(* CODESYS project PlantaFinal.project

Project tree, tasks and I/O mapping:
  Device : CODESYS Control Win V3, 3S - Smart Software Solutions GmbH, order no. 305021, version 3.5.8.10
    application Application
      libraries: Standard, * (System)
      task MainTask (cyclic, interval t#20ms, priority 1) calls PLC_PRG
      program PLC_PRG [LD]
      Symbols
*)

// Device/Application/PLC_PRG
PROGRAM PLC_PRG
VAR
	//Entradas - Gerais
	_EmergencyStop: BOOL;
	_Reset: BOOL;
	_Start: BOOL;
	_Stop: BOOL;
	_Auto: BOOL;
	_Manual: BOOL;
	
	//Entradas - Stage 01
	_S01_VisionSensor1: WORD;
	_S01_VisionSensor2: WORD;	
	_S01_Sensor1: BOOL;
	_S01_Sensor2: BOOL;	
	_S01_Pusher1Back: BOOL;
	_S01_Pusher2Back: BOOL;	
	_S01_Pusher1Front: BOOL;
	_S01_Pusher2Front: BOOL;	
	_S01_AtPusher1Exit: BOOL;
	_S01_AtPusher2Exit: BOOL;
	_S01_LidAtExit: BOOL;
	_S01_BaseAtExit: BOOL;
	
	//Entradas - Stage 02
	_S02_LidAtEntry: BOOL;
	_S02_BaseAtEntry: BOOL;
	_S02_LidAtPlace: BOOL;
	_S02_LidClamped: BOOL;
	_S02_BaseClamped: BOOL;
	_S02_MovingZ: BOOL;
	_S02_BaseAtPlace: BOOL;
	_S02_MovingX: BOOL;
	_S02_PartLeaving: BOOL;
	
	//Entradas - Stage 03
	_S03_ItemAtEntry: BOOL;
	_S03_ItemADetected: BOOL;
	_S03_MovingX: BOOL;
	_S03_MovingZ: BOOL;
	
	//Entradas - Stage 04
	_S04_AtEntry: BOOL;
	_S04_AtLoad: BOOL;
	_S04_AtLeft: BOOL;
	_S04_AtRight: BOOL;
	_S04_AtMiddle: BOOL;
	_S04_MovingZ: BOOL;
	_S04_MovingX: BOOL;
	
	//Saidas - Gerais
	StopLight: BOOL;
	StartLight: BOOL;
	ResetLight: BOOL;
	ProductCounter: WORD;
	
	//Saidas - Stage 01
	S01_EntryConveyor1: BOOL;
	S01_EntryConveyor2: BOOL;
	S01_Conveyor1: BOOL;
	S01_Conveyor2: BOOL;
	S01_Pusher1: BOOL;
	S01_Pusher2: BOOL;
	S01_RollerStop1: BOOL;
	S01_RollerStop2: BOOL;
	
	//Saidas - Stage 02
	S02_LidsConveyor: BOOL;
	S02_BasesConveyor: BOOL;
	S02_ClampLid: BOOL;
	S02_MoveZ: BOOL;
	S02_MoveX: BOOL;
	S02_Grab: BOOL;
	S02_ClampBase: BOOL;
	S02_PosRaiseBase: BOOL;
	
	//Saidas - Stage 03
	S03_Grab: BOOL;
	S03_MoveZ: BOOL;
	S03_MoveX: BOOL;
	S03_EntryConveyor: BOOL;
	S03_Emitter: BOOL;
	S03_RollerConveyor: BOOL;

	//Saidas - Stage 03
	S04_EntryConveyor: BOOL;	
	S04_LoadConveyor: BOOL;
	S04_ForksLeft: BOOL;
	S04_ForksRight: BOOL;
	S04_Lift: BOOL;	
	S04_TargetPosition: INT;	
	
	//Sinais - Gerais
	Enable: BOOL;
	Stopping: BOOL;
	OnDelay: TON;
	OffDelay: TOF;
	AutoMode: BOOL;
	ManualMode: BOOL;	
	Caso: INT;	
	BaseAzul: WORD :=3;
	BaseVerde: WORD :=6;
	TampaAzul: WORD :=2;
	TampaVerde: WORD :=5;
	
	//Sinais - Stage 01
	S01_MX10: BOOL;
	S01_MX11: BOOL;
	S01_MX12: BOOL;
	S01_MX13: BOOL;
	S01_MX14: BOOL;
	S01_MX15: BOOL;
	S01_MX16: BOOL;
	S01_MX17: BOOL;
	F_TRIG_0: F_TRIG;
	F_TRIG_1: F_TRIG;
	F_TRIG_2: F_TRIG;
	F_TRIG_3: F_TRIG;
	F_TRIG_4: F_TRIG;	
	F_TRIG_5: F_TRIG;
	F_TRIG_6: F_TRIG;
	F_TRIG_7: F_TRIG;
	F_TRIG_8: F_TRIG;
	PartsAtExit: BOOL;
	TON_1: TON;
	TON_2: TON;
	TON_3: TON;
	TON_4: TON;
	TON_5: TON;
	
	//Sinais - Stage 02
	S02_MX00: BOOL;
	S02_MX01: BOOL;
	TON_0: TON;
	S02_BaseAtS02: BOOL;
	S02_LidAtS02: BOOL;	
	S02_MX02: BOOL;
	S02_MX20: BOOL;
	S02_MX21: BOOL;
	S02_MX10: BOOL;
	S02_MX11: BOOL;
	F_TRIG_9: F_TRIG;
	S02_MX12: BOOL;
	F_TRIG_10: F_TRIG;
	S02_MX13: BOOL;
	F_TRIG_11: F_TRIG;
	S02_MX14: BOOL;
	F_TRIG_12: F_TRIG;
	S02_MX15: BOOL;
	F_TRIG_13: F_TRIG;
	S02_MX16: BOOL;
	F_TRIG_14: F_TRIG;
	ProductDone: BOOL;
	
	//Sinais - Stage 03
	S03_MX00: BOOL;
	S03_MX01: BOOL;
	F_TRIG_15: F_TRIG;
	S03_MX02: BOOL;
	F_TRIG_16: F_TRIG;
	F_TRIG_17: F_TRIG;
	S03_MX03: BOOL;
	F_TRIG_18: F_TRIG;
	S03_MX04: BOOL;
	S03_MX05: BOOL;
	F_TRIG_19: F_TRIG;
	S03_MX06: BOOL;
	F_TRIG_20: F_TRIG;
	S03_MX07: BOOL;
	F_TRIG_21: F_TRIG;
	S03_MX08: BOOL;
	S03_MX09: BOOL;
	F_TRIG_22: F_TRIG;
	
	//Sinais - Stage 04
	S04_MX10: BOOL;
	S04_MX11: BOOL;
	S04_MX12: BOOL;
	S04_MX13: BOOL;
	CTU_0: CTU;
	Contagem: INT;
	Q: BOOL;
	S04_MX14: BOOL;
	S04_MX15: BOOL;
	R_TRIG_0: R_TRIG;
	R_TRIG_1: R_TRIG;
	
END_VAR
VAR // added by the converter: edge detectors and wires of the graphical bodies
    _w1, _w2, _w3, _w4, _w5, _w6, _w7, _w8, _w9, _w10, _w11, _w12, _w13, _w14, _w15, _w16, _w17, _w18, _w19, _w20, _w21, _w22, _w23, _w24, _w25, _w26, _w27, _w28, _w29, _w30, _w31, _w32, _w33, _w34, _w35, _w36, _w37, _w38, _w39, _w40, _w41, _w42, _w43, _w44, _w45, _w46, _w47, _w48, _w49, _w50, _w51, _w52, _w53, _w54, _w55, _w56, _w57, _w58, _w59, _w60, _w61, _w62, _w63, _w64, _w65, _w66, _w67, _w68 : BOOL;
    _rt1, _rt2, _rt3, _rt4, _rt5, _rt6, _rt7, _rt8 : R_TRIG;
    _ft1, _ft2, _ft3, _ft4, _ft5, _ft6, _ft7, _ft8, _ft9, _ft10, _ft11, _ft12, _ft13, _ft14, _ft15 : F_TRIG;
END_VAR

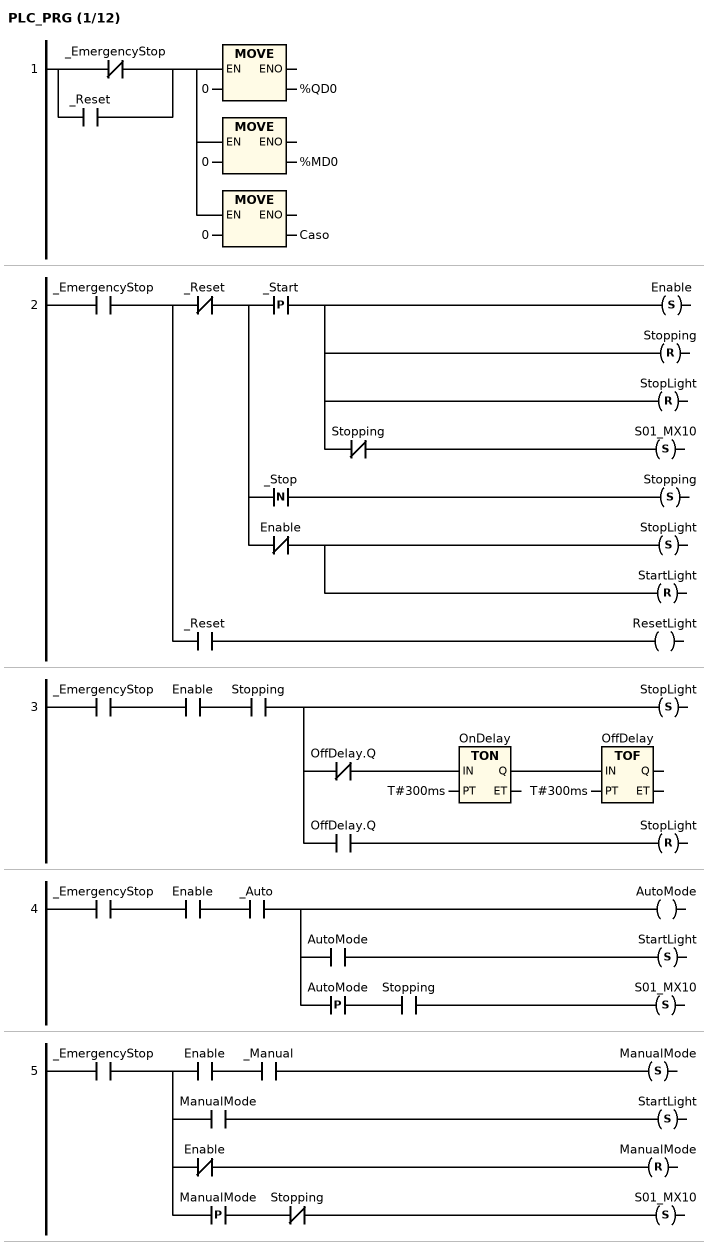
// NETWORK 1
_w1 := NOT _EmergencyStop OR _Reset;
IF _w1 THEN %QD0 := 0; END_IF
IF _w1 THEN %MD0 := 0; END_IF
IF _w1 THEN Caso := 0; END_IF

// NETWORK 2
_w2 := _EmergencyStop AND NOT _Reset;
_rt1(CLK := _Start);
_w3 := _w2 AND _rt1.Q;
Enable S= _w3;
Stopping R= _w3;
StopLight R= _w3;
S01_MX10 S= _w3 AND NOT Stopping;
_ft1(CLK := _Stop);
Stopping S= _w2 AND _ft1.Q;
_w4 := _w2 AND NOT Enable;
StopLight S= _w4;
StartLight R= _w4;
ResetLight := _EmergencyStop AND _Reset;

// NETWORK 3
_w5 := _EmergencyStop AND Enable AND Stopping;
StopLight S= _w5;
OnDelay(IN := _w5 AND NOT OffDelay.Q, PT := T#300ms); // TON
OffDelay(IN := OnDelay.Q, PT := T#300ms); // TOF
StopLight R= _w5 AND OffDelay.Q;

// NETWORK 4
_w6 := _EmergencyStop AND Enable AND _Auto;
AutoMode := _w6;
StartLight S= _w6 AND AutoMode;
_rt2(CLK := AutoMode);
S01_MX10 S= _w6 AND _rt2.Q AND Stopping;

// NETWORK 5
ManualMode S= _EmergencyStop AND Enable AND _Manual;
StartLight S= _EmergencyStop AND ManualMode;
ManualMode R= _EmergencyStop AND NOT Enable;
_rt3(CLK := ManualMode);
S01_MX10 S= _EmergencyStop AND _rt3.Q AND NOT Stopping;

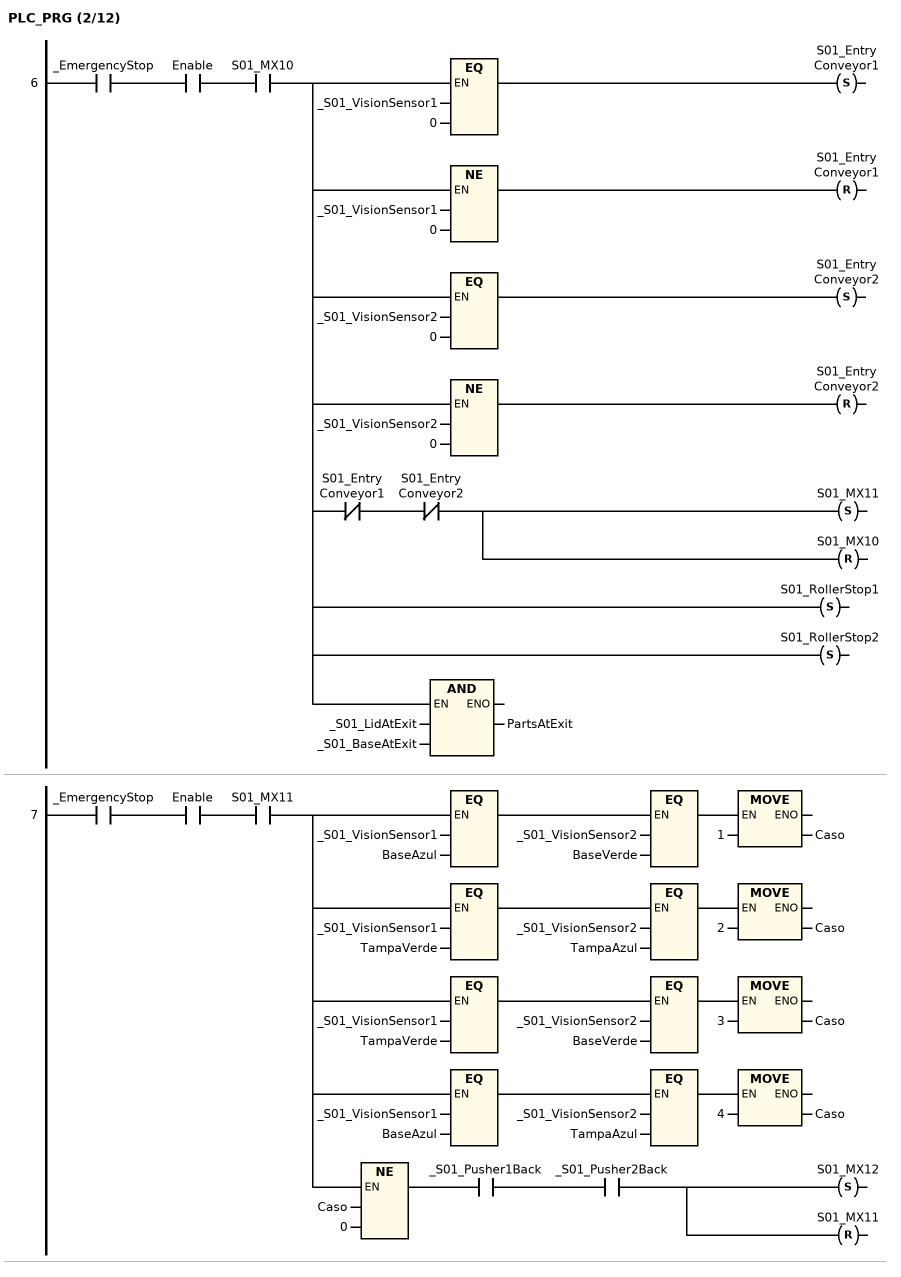
// NETWORK 6
_w7 := _EmergencyStop AND Enable AND S01_MX10;
S01_EntryConveyor1 S= _w7 AND _S01_VisionSensor1 = 0;
S01_EntryConveyor1 R= _w7 AND _S01_VisionSensor1 <> 0;
S01_EntryConveyor2 S= _w7 AND _S01_VisionSensor2 = 0;
S01_EntryConveyor2 R= _w7 AND _S01_VisionSensor2 <> 0;
_w8 := _w7 AND NOT S01_EntryConveyor1 AND NOT S01_EntryConveyor2;
S01_MX11 S= _w8;
S01_MX10 R= _w8;
S01_RollerStop1 S= _w7;
S01_RollerStop2 S= _w7;
IF _w7 THEN PartsAtExit := _S01_LidAtExit AND _S01_BaseAtExit; END_IF

// NETWORK 7
_w9 := _EmergencyStop AND Enable AND S01_MX11;
IF _w9 AND _S01_VisionSensor1 = BaseAzul AND _S01_VisionSensor2 = BaseVerde THEN Caso := 1; END_IF
IF _w9 AND _S01_VisionSensor1 = TampaVerde AND _S01_VisionSensor2 = TampaAzul THEN Caso := 2; END_IF
IF _w9 AND _S01_VisionSensor1 = TampaVerde AND _S01_VisionSensor2 = BaseVerde THEN Caso := 3; END_IF
IF _w9 AND _S01_VisionSensor1 = BaseAzul AND _S01_VisionSensor2 = TampaAzul THEN Caso := 4; END_IF
_w10 := (_w9 AND Caso <> 0) AND _S01_Pusher1Back AND _S01_Pusher2Back;
S01_MX12 S= _w10;
S01_MX11 R= _w10;

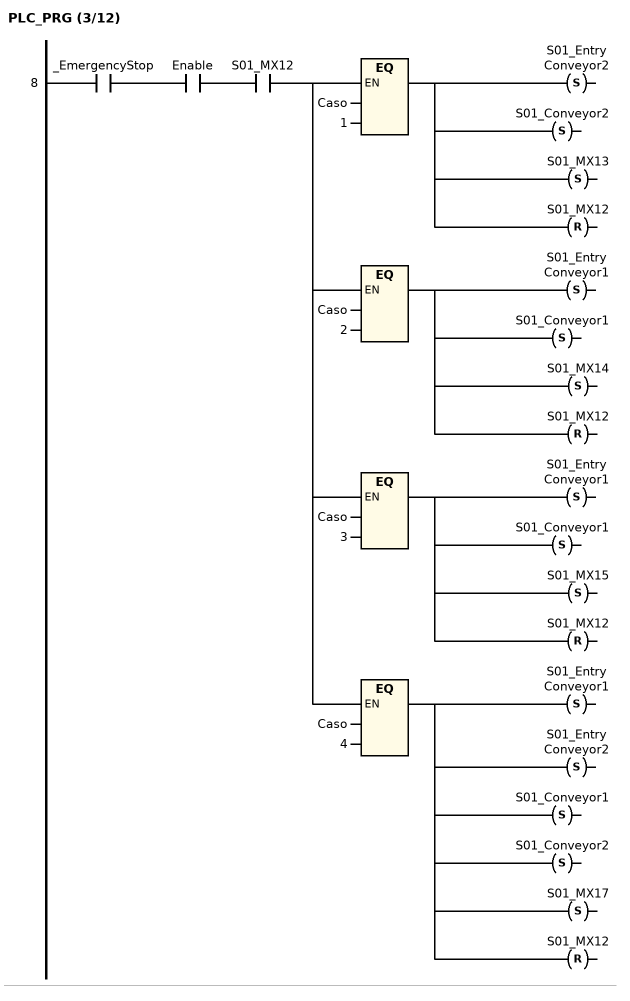
// NETWORK 8
_w11 := _EmergencyStop AND Enable AND S01_MX12;
_w12 := _w11 AND Caso = 1;
S01_EntryConveyor2 S= _w12;
S01_Conveyor2 S= _w12;
S01_MX13 S= _w12;
S01_MX12 R= _w12;
_w13 := _w11 AND Caso = 2;
S01_EntryConveyor1 S= _w13;
S01_Conveyor1 S= _w13;
S01_MX14 S= _w13;
S01_MX12 R= _w13;
_w14 := _w11 AND Caso = 3;
S01_EntryConveyor1 S= _w14;
S01_Conveyor1 S= _w14;
S01_MX15 S= _w14;
S01_MX12 R= _w14;
_w15 := _w11 AND Caso = 4;
S01_EntryConveyor1 S= _w15;
S01_EntryConveyor2 S= _w15;
S01_Conveyor1 S= _w15;
S01_Conveyor2 S= _w15;
S01_MX17 S= _w15;
S01_MX12 R= _w15;

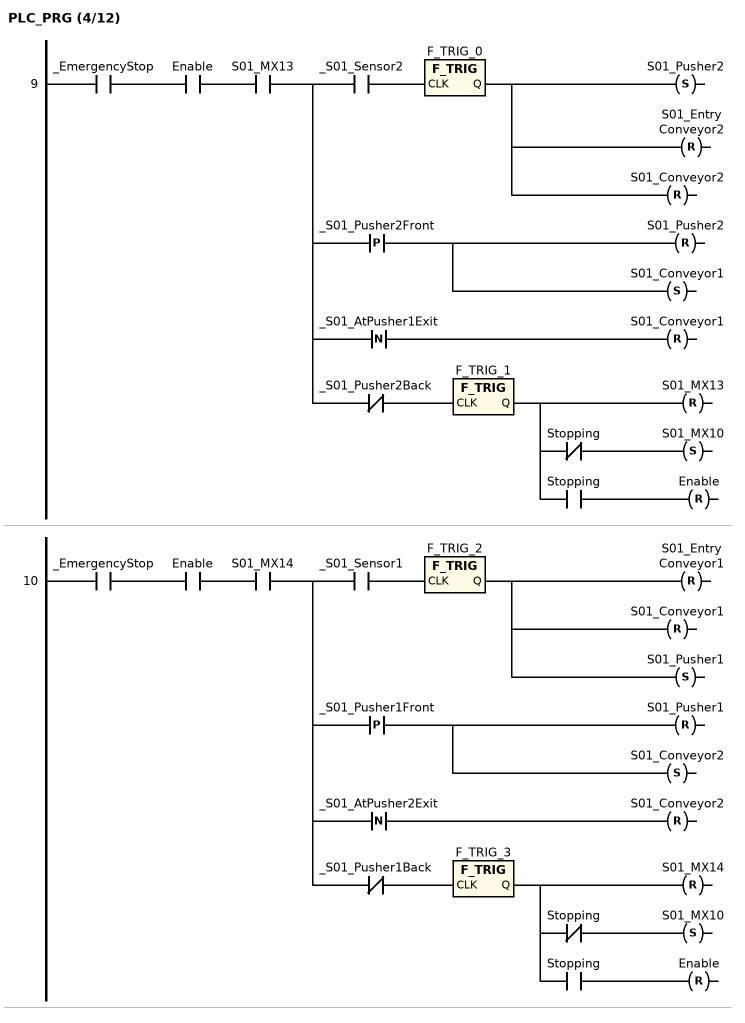
// NETWORK 9
_w16 := _EmergencyStop AND Enable AND S01_MX13;
F_TRIG_0(CLK := _w16 AND _S01_Sensor2); // F_TRIG
S01_Pusher2 S= F_TRIG_0.Q;
S01_EntryConveyor2 R= F_TRIG_0.Q;
S01_Conveyor2 R= F_TRIG_0.Q;
_rt4(CLK := _S01_Pusher2Front);
_w17 := _w16 AND _rt4.Q;
S01_Pusher2 R= _w17;
S01_Conveyor1 S= _w17;
_ft2(CLK := _S01_AtPusher1Exit);
S01_Conveyor1 R= _w16 AND _ft2.Q;
F_TRIG_1(CLK := _w16 AND NOT _S01_Pusher2Back); // F_TRIG
S01_MX13 R= F_TRIG_1.Q;
S01_MX10 S= F_TRIG_1.Q AND NOT Stopping;
Enable R= F_TRIG_1.Q AND Stopping;

// NETWORK 10
_w18 := _EmergencyStop AND Enable AND S01_MX14;
F_TRIG_2(CLK := _w18 AND _S01_Sensor1); // F_TRIG
S01_EntryConveyor1 R= F_TRIG_2.Q;
S01_Conveyor1 R= F_TRIG_2.Q;
S01_Pusher1 S= F_TRIG_2.Q;
_rt5(CLK := _S01_Pusher1Front);
_w19 := _w18 AND _rt5.Q;
S01_Pusher1 R= _w19;
S01_Conveyor2 S= _w19;
_ft3(CLK := _S01_AtPusher2Exit);
S01_Conveyor2 R= _w18 AND _ft3.Q;
F_TRIG_3(CLK := _w18 AND NOT _S01_Pusher1Back); // F_TRIG
S01_MX14 R= F_TRIG_3.Q;
S01_MX10 S= F_TRIG_3.Q AND NOT Stopping;
Enable R= F_TRIG_3.Q AND Stopping;

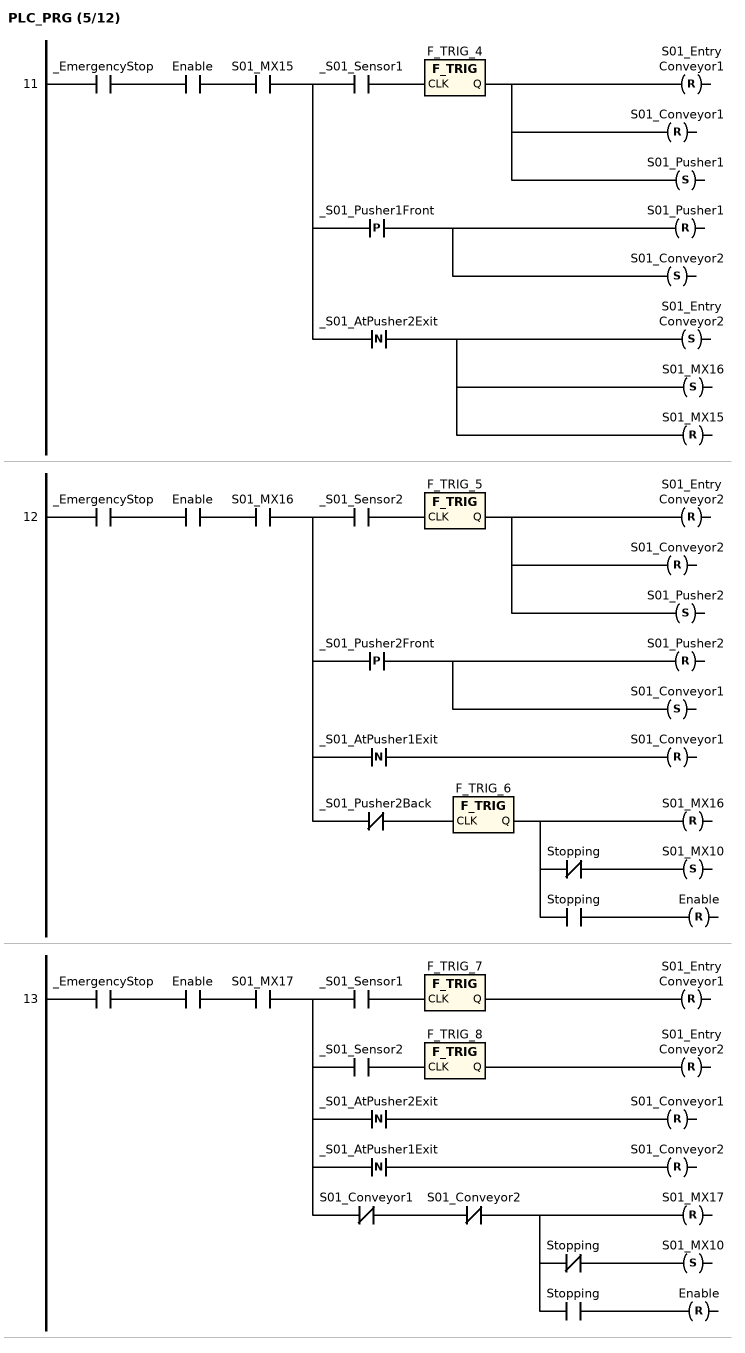
// NETWORK 11
_w20 := _EmergencyStop AND Enable AND S01_MX15;
F_TRIG_4(CLK := _w20 AND _S01_Sensor1); // F_TRIG
S01_EntryConveyor1 R= F_TRIG_4.Q;
S01_Conveyor1 R= F_TRIG_4.Q;
S01_Pusher1 S= F_TRIG_4.Q;
_rt6(CLK := _S01_Pusher1Front);
_w21 := _w20 AND _rt6.Q;
S01_Pusher1 R= _w21;
S01_Conveyor2 S= _w21;
_ft4(CLK := _S01_AtPusher2Exit);
_w22 := _w20 AND _ft4.Q;
S01_EntryConveyor2 S= _w22;
S01_MX16 S= _w22;
S01_MX15 R= _w22;

// NETWORK 12
_w23 := _EmergencyStop AND Enable AND S01_MX16;
F_TRIG_5(CLK := _w23 AND _S01_Sensor2); // F_TRIG
S01_EntryConveyor2 R= F_TRIG_5.Q;
S01_Conveyor2 R= F_TRIG_5.Q;
S01_Pusher2 S= F_TRIG_5.Q;
_rt7(CLK := _S01_Pusher2Front);
_w24 := _w23 AND _rt7.Q;
S01_Pusher2 R= _w24;
S01_Conveyor1 S= _w24;
_ft5(CLK := _S01_AtPusher1Exit);
S01_Conveyor1 R= _w23 AND _ft5.Q;
F_TRIG_6(CLK := _w23 AND NOT _S01_Pusher2Back); // F_TRIG
S01_MX16 R= F_TRIG_6.Q;
S01_MX10 S= F_TRIG_6.Q AND NOT Stopping;
Enable R= F_TRIG_6.Q AND Stopping;

// NETWORK 13
_w25 := _EmergencyStop AND Enable AND S01_MX17;
F_TRIG_7(CLK := _w25 AND _S01_Sensor1); // F_TRIG
S01_EntryConveyor1 R= F_TRIG_7.Q;
F_TRIG_8(CLK := _w25 AND _S01_Sensor2); // F_TRIG
S01_EntryConveyor2 R= F_TRIG_8.Q;
_ft6(CLK := _S01_AtPusher2Exit);
S01_Conveyor1 R= _w25 AND _ft6.Q;
_ft7(CLK := _S01_AtPusher1Exit);
S01_Conveyor2 R= _w25 AND _ft7.Q;
_w26 := _w25 AND NOT S01_Conveyor1 AND NOT S01_Conveyor2;
S01_MX17 R= _w26;
S01_MX10 S= _w26 AND NOT Stopping;
Enable R= _w26 AND Stopping;

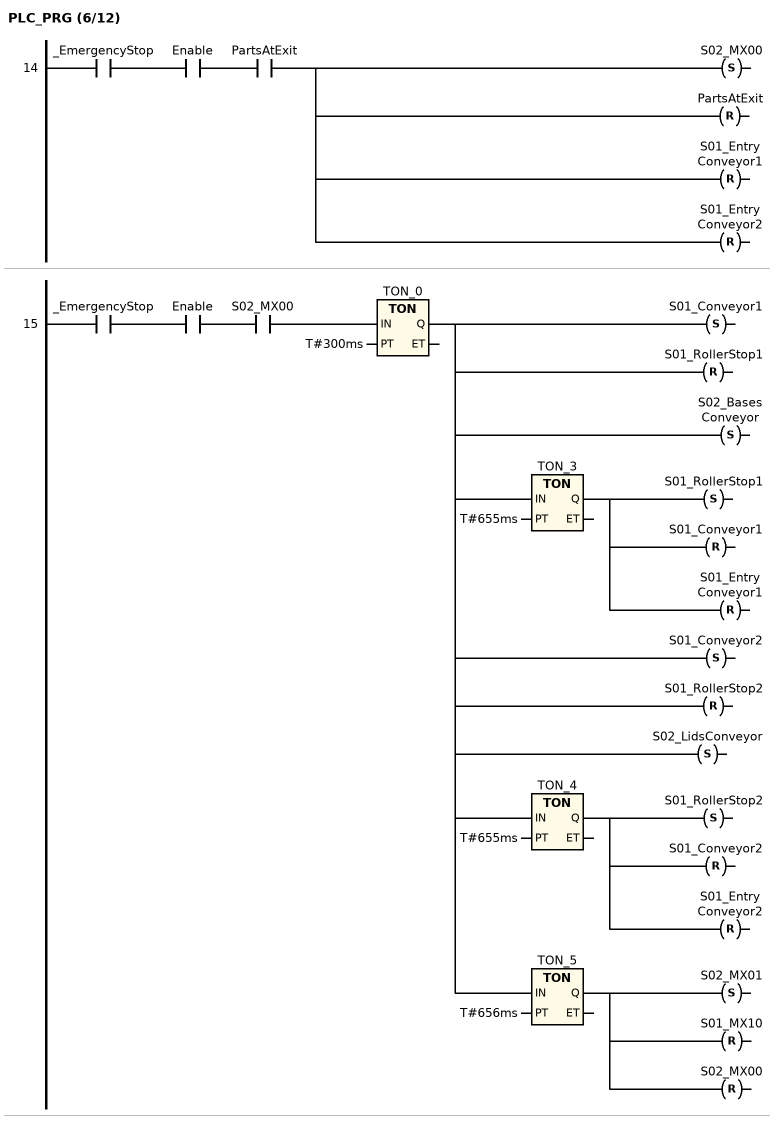
// NETWORK 14
_w27 := _EmergencyStop AND Enable AND PartsAtExit;
S02_MX00 S= _w27;
PartsAtExit R= _w27;
S01_EntryConveyor1 R= _w27;
S01_EntryConveyor2 R= _w27;

// NETWORK 15
TON_0(IN := _EmergencyStop AND Enable AND S02_MX00, PT := T#300ms); // TON
S01_Conveyor1 S= TON_0.Q;
S01_RollerStop1 R= TON_0.Q;
S02_BasesConveyor S= TON_0.Q;
TON_3(IN := TON_0.Q, PT := T#655ms); // TON
S01_RollerStop1 S= TON_3.Q;
S01_Conveyor1 R= TON_3.Q;
S01_EntryConveyor1 R= TON_3.Q;
S01_Conveyor2 S= TON_0.Q;
S01_RollerStop2 R= TON_0.Q;
S02_LidsConveyor S= TON_0.Q;
TON_4(IN := TON_0.Q, PT := T#655ms); // TON
S01_RollerStop2 S= TON_4.Q;
S01_Conveyor2 R= TON_4.Q;
S01_EntryConveyor2 R= TON_4.Q;
TON_5(IN := TON_0.Q, PT := T#656ms); // TON
S02_MX01 S= TON_5.Q;
S01_MX10 R= TON_5.Q;
S02_MX00 R= TON_5.Q;

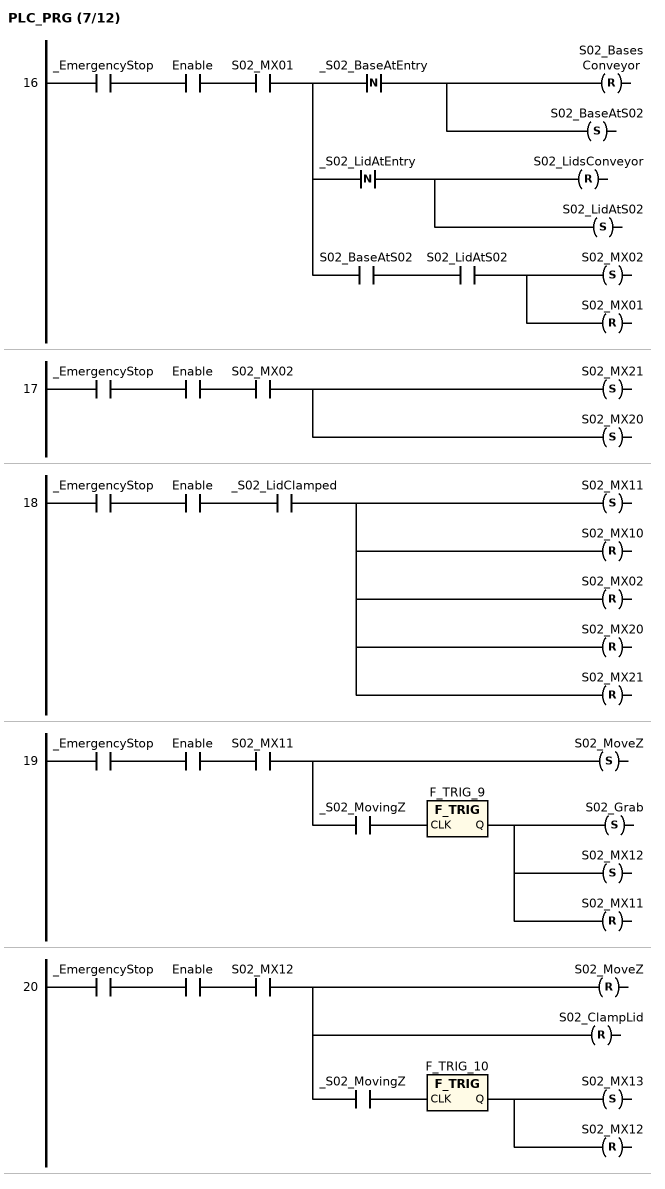
// NETWORK 16
_w28 := _EmergencyStop AND Enable AND S02_MX01;
_ft8(CLK := _S02_BaseAtEntry);
_w29 := _w28 AND _ft8.Q;
S02_BasesConveyor R= _w29;
S02_BaseAtS02 S= _w29;
_ft9(CLK := _S02_LidAtEntry);
_w30 := _w28 AND _ft9.Q;
S02_LidsConveyor R= _w30;
S02_LidAtS02 S= _w30;
_w31 := _w28 AND S02_BaseAtS02 AND S02_LidAtS02;
S02_MX02 S= _w31;
S02_MX01 R= _w31;

// NETWORK 17
_w32 := _EmergencyStop AND Enable AND S02_MX02;
S02_MX21 S= _w32;
S02_MX20 S= _w32;

// NETWORK 18
_w33 := _EmergencyStop AND Enable AND _S02_LidClamped;
S02_MX11 S= _w33;
S02_MX10 R= _w33;
S02_MX02 R= _w33;
S02_MX20 R= _w33;
S02_MX21 R= _w33;

// NETWORK 19
_w34 := _EmergencyStop AND Enable AND S02_MX11;
S02_MoveZ S= _w34;
F_TRIG_9(CLK := _w34 AND _S02_MovingZ); // F_TRIG
S02_Grab S= F_TRIG_9.Q;
S02_MX12 S= F_TRIG_9.Q;
S02_MX11 R= F_TRIG_9.Q;

// NETWORK 20
_w35 := _EmergencyStop AND Enable AND S02_MX12;
S02_MoveZ R= _w35;
S02_ClampLid R= _w35;
F_TRIG_10(CLK := _w35 AND _S02_MovingZ); // F_TRIG
S02_MX13 S= F_TRIG_10.Q;
S02_MX12 R= F_TRIG_10.Q;

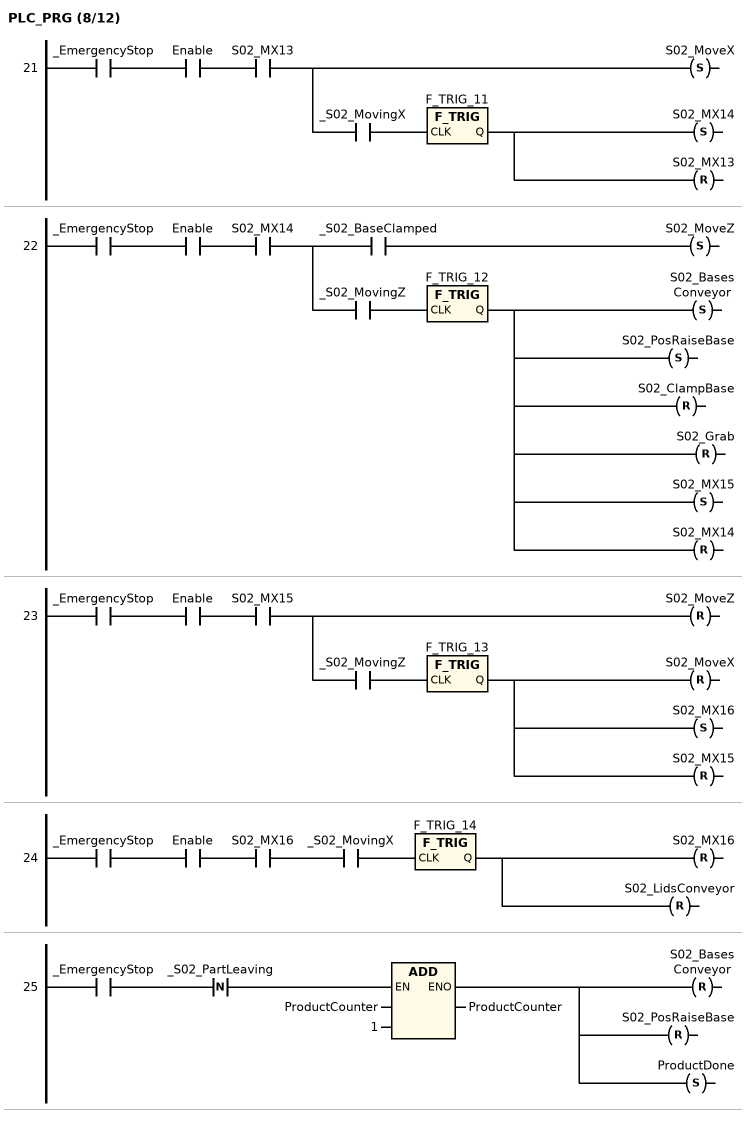
// NETWORK 21
_w36 := _EmergencyStop AND Enable AND S02_MX13;
S02_MoveX S= _w36;
F_TRIG_11(CLK := _w36 AND _S02_MovingX); // F_TRIG
S02_MX14 S= F_TRIG_11.Q;
S02_MX13 R= F_TRIG_11.Q;

// NETWORK 22
_w37 := _EmergencyStop AND Enable AND S02_MX14;
S02_MoveZ S= _w37 AND _S02_BaseClamped;
F_TRIG_12(CLK := _w37 AND _S02_MovingZ); // F_TRIG
S02_BasesConveyor S= F_TRIG_12.Q;
S02_PosRaiseBase S= F_TRIG_12.Q;
S02_ClampBase R= F_TRIG_12.Q;
S02_Grab R= F_TRIG_12.Q;
S02_MX15 S= F_TRIG_12.Q;
S02_MX14 R= F_TRIG_12.Q;

// NETWORK 23
_w38 := _EmergencyStop AND Enable AND S02_MX15;
S02_MoveZ R= _w38;
F_TRIG_13(CLK := _w38 AND _S02_MovingZ); // F_TRIG
S02_MoveX R= F_TRIG_13.Q;
S02_MX16 S= F_TRIG_13.Q;
S02_MX15 R= F_TRIG_13.Q;

// NETWORK 24
F_TRIG_14(CLK := _EmergencyStop AND Enable AND S02_MX16 AND _S02_MovingX); // F_TRIG
S02_MX16 R= F_TRIG_14.Q;
S02_LidsConveyor R= F_TRIG_14.Q;

// NETWORK 25
_ft10(CLK := _S02_PartLeaving);
_w39 := _EmergencyStop AND _ft10.Q;
IF _w39 THEN ProductCounter := ProductCounter + 1; END_IF
S02_BasesConveyor R= _w39;
S02_PosRaiseBase R= _w39;
ProductDone S= _w39;

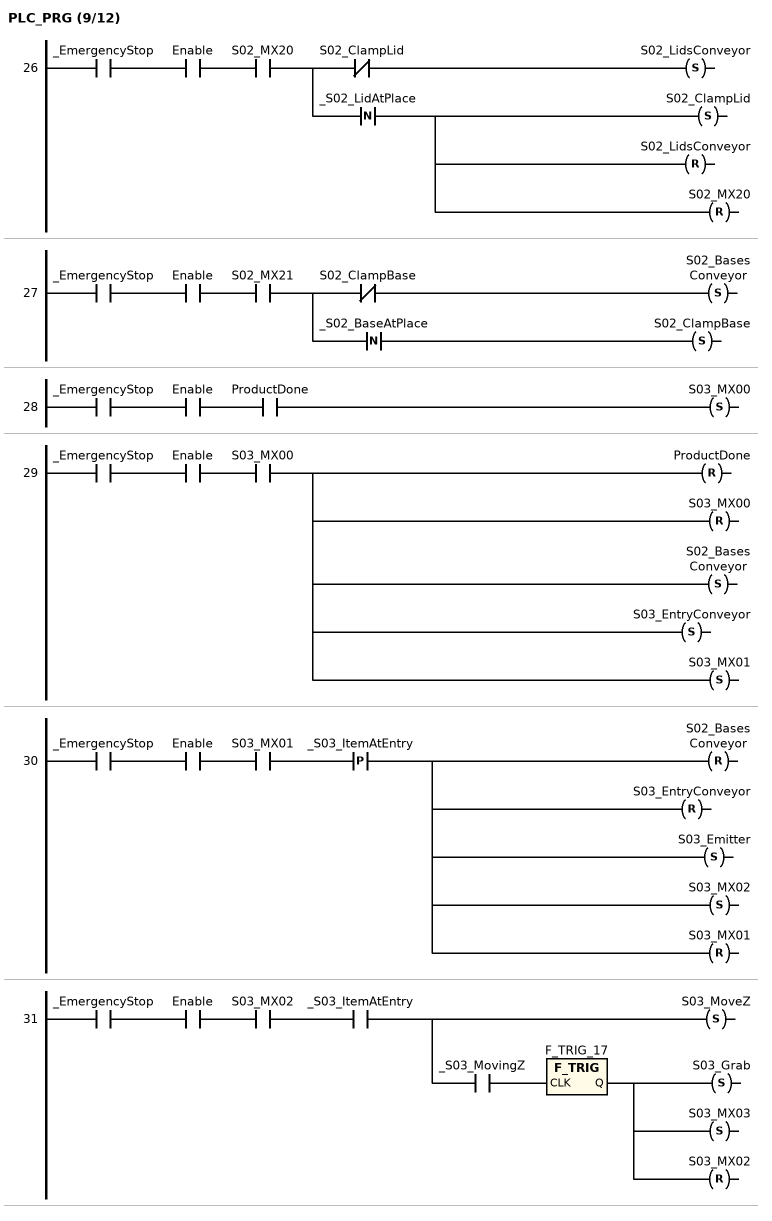
// NETWORK 26
_w40 := _EmergencyStop AND Enable AND S02_MX20;
S02_LidsConveyor S= _w40 AND NOT S02_ClampLid;
_ft11(CLK := _S02_LidAtPlace);
_w41 := _w40 AND _ft11.Q;
S02_ClampLid S= _w41;
S02_LidsConveyor R= _w41;
S02_MX20 R= _w41;

// NETWORK 27
_w42 := _EmergencyStop AND Enable AND S02_MX21;
S02_BasesConveyor S= _w42 AND NOT S02_ClampBase;
_ft12(CLK := _S02_BaseAtPlace);
S02_ClampBase S= _w42 AND _ft12.Q;

// NETWORK 28
S03_MX00 S= _EmergencyStop AND Enable AND ProductDone;

// NETWORK 29
_w43 := _EmergencyStop AND Enable AND S03_MX00;
ProductDone R= _w43;
S03_MX00 R= _w43;
S02_BasesConveyor S= _w43;
S03_EntryConveyor S= _w43;
S03_MX01 S= _w43;

// NETWORK 30
_rt8(CLK := _S03_ItemAtEntry);
_w44 := _EmergencyStop AND Enable AND S03_MX01 AND _rt8.Q;
S02_BasesConveyor R= _w44;
S03_EntryConveyor R= _w44;
S03_Emitter S= _w44;
S03_MX02 S= _w44;
S03_MX01 R= _w44;

// NETWORK 31
_w45 := _EmergencyStop AND Enable AND S03_MX02 AND _S03_ItemAtEntry;
S03_MoveZ S= _w45;
F_TRIG_17(CLK := _w45 AND _S03_MovingZ); // F_TRIG
S03_Grab S= F_TRIG_17.Q;
S03_MX03 S= F_TRIG_17.Q;
S03_MX02 R= F_TRIG_17.Q;

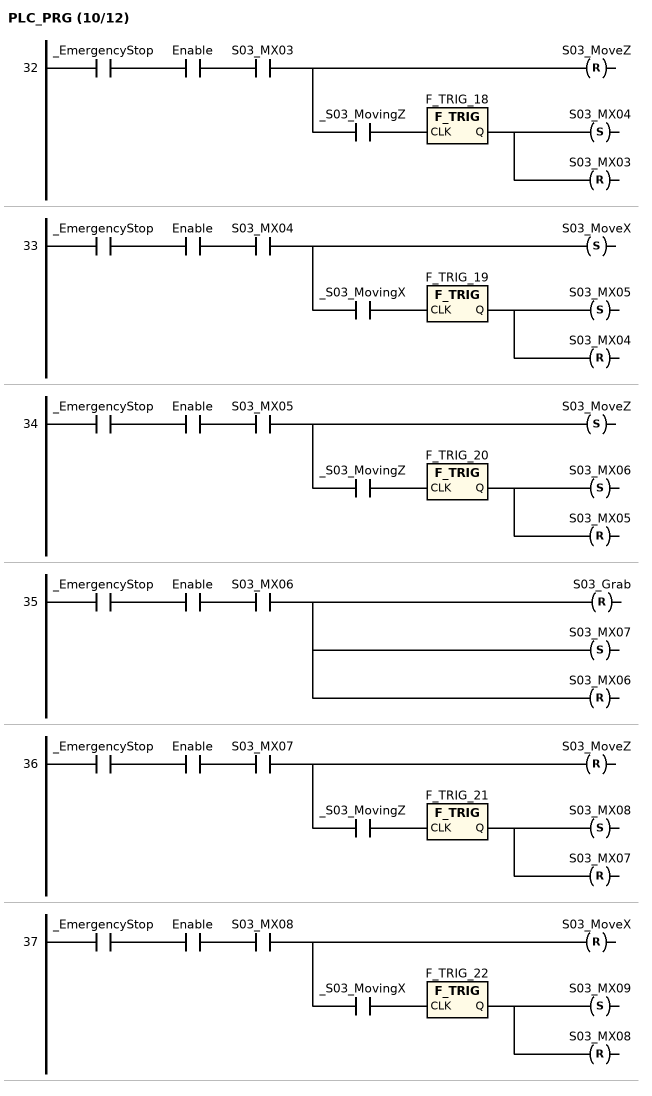
// NETWORK 32
_w46 := _EmergencyStop AND Enable AND S03_MX03;
S03_MoveZ R= _w46;
F_TRIG_18(CLK := _w46 AND _S03_MovingZ); // F_TRIG
S03_MX04 S= F_TRIG_18.Q;
S03_MX03 R= F_TRIG_18.Q;

// NETWORK 33
_w47 := _EmergencyStop AND Enable AND S03_MX04;
S03_MoveX S= _w47;
F_TRIG_19(CLK := _w47 AND _S03_MovingX); // F_TRIG
S03_MX05 S= F_TRIG_19.Q;
S03_MX04 R= F_TRIG_19.Q;

// NETWORK 34
_w48 := _EmergencyStop AND Enable AND S03_MX05;
S03_MoveZ S= _w48;
F_TRIG_20(CLK := _w48 AND _S03_MovingZ); // F_TRIG
S03_MX06 S= F_TRIG_20.Q;
S03_MX05 R= F_TRIG_20.Q;

// NETWORK 35
_w49 := _EmergencyStop AND Enable AND S03_MX06;
S03_Grab R= _w49;
S03_MX07 S= _w49;
S03_MX06 R= _w49;

// NETWORK 36
_w50 := _EmergencyStop AND Enable AND S03_MX07;
S03_MoveZ R= _w50;
F_TRIG_21(CLK := _w50 AND _S03_MovingZ); // F_TRIG
S03_MX08 S= F_TRIG_21.Q;
S03_MX07 R= F_TRIG_21.Q;

// NETWORK 37
_w51 := _EmergencyStop AND Enable AND S03_MX08;
S03_MoveX R= _w51;
F_TRIG_22(CLK := _w51 AND _S03_MovingX); // F_TRIG
S03_MX09 S= F_TRIG_22.Q;
S03_MX08 R= F_TRIG_22.Q;

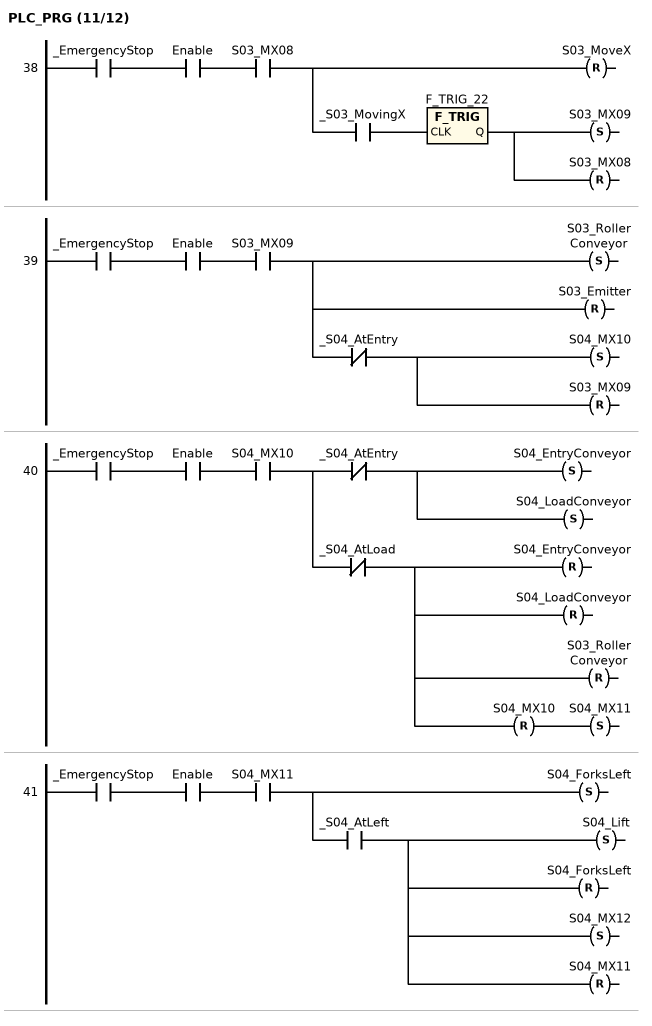
// NETWORK 38
_w52 := _EmergencyStop AND Enable AND S03_MX08;
S03_MoveX R= _w52;
F_TRIG_22(CLK := _w52 AND _S03_MovingX); // F_TRIG
S03_MX09 S= F_TRIG_22.Q;
S03_MX08 R= F_TRIG_22.Q;

// NETWORK 39
_w53 := _EmergencyStop AND Enable AND S03_MX09;
S03_RollerConveyor S= _w53;
S03_Emitter R= _w53;
_w54 := _w53 AND NOT _S04_AtEntry;
S04_MX10 S= _w54;
S03_MX09 R= _w54;

// NETWORK 40
_w55 := _EmergencyStop AND Enable AND S04_MX10;
_w56 := _w55 AND NOT _S04_AtEntry;
S04_EntryConveyor S= _w56;
S04_LoadConveyor S= _w56;
_w57 := _w55 AND NOT _S04_AtLoad;
S04_EntryConveyor R= _w57;
S04_LoadConveyor R= _w57;
S03_RollerConveyor R= _w57;
S04_MX10 R= _w57;
S04_MX11 S= _w57;

// NETWORK 41
_w58 := _EmergencyStop AND Enable AND S04_MX11;
S04_ForksLeft S= _w58;
_w59 := _w58 AND _S04_AtLeft;
S04_Lift S= _w59;
S04_ForksLeft R= _w59;
S04_MX12 S= _w59;
S04_MX11 R= _w59;

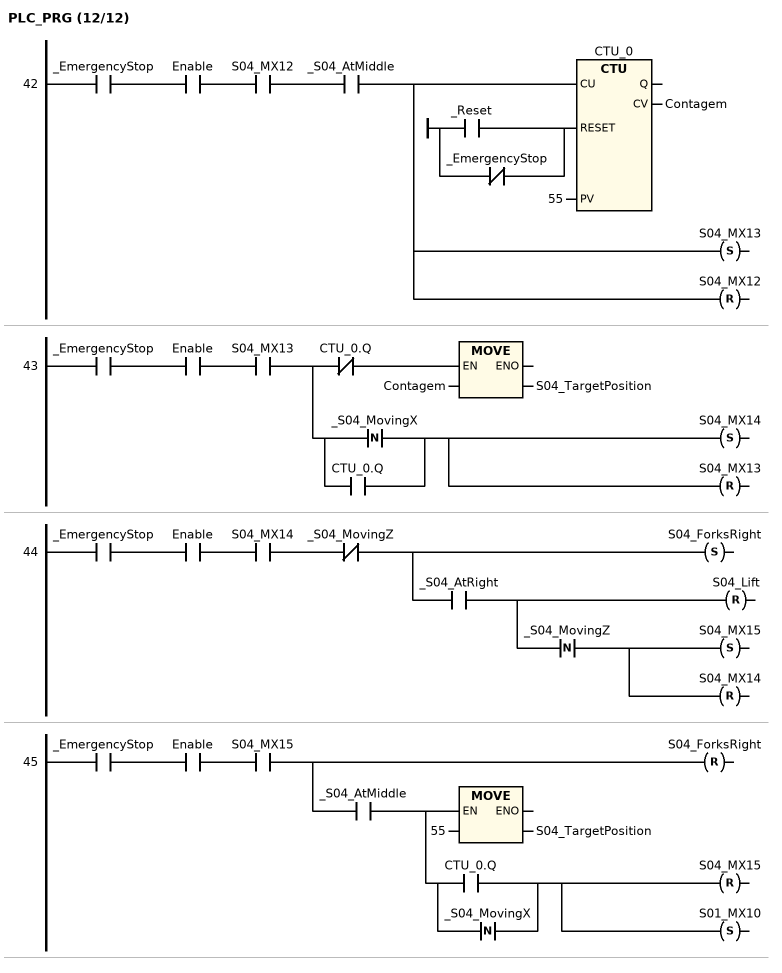
// NETWORK 42
_w60 := _EmergencyStop AND Enable AND S04_MX12 AND _S04_AtMiddle;
CTU_0(CU := _w60, RESET := _Reset OR NOT _EmergencyStop, PV := 55, CV => Contagem); // CTU
S04_MX13 S= _w60;
S04_MX12 R= _w60;

// NETWORK 43
_w61 := _EmergencyStop AND Enable AND S04_MX13;
IF _w61 AND NOT CTU_0.Q THEN S04_TargetPosition := Contagem; END_IF
_ft13(CLK := _S04_MovingX);
_w62 := _w61 AND (_ft13.Q OR CTU_0.Q);
S04_MX14 S= _w62;
S04_MX13 R= _w62;

// NETWORK 44
_w63 := _EmergencyStop AND Enable AND S04_MX14 AND NOT _S04_MovingZ;
S04_ForksRight S= _w63;
_w64 := _w63 AND _S04_AtRight;
S04_Lift R= _w64;
_ft14(CLK := _S04_MovingZ);
_w65 := _w64 AND _ft14.Q;
S04_MX15 S= _w65;
S04_MX14 R= _w65;

// NETWORK 45
_w66 := _EmergencyStop AND Enable AND S04_MX15;
S04_ForksRight R= _w66;
_w67 := _w66 AND _S04_AtMiddle;
IF _w67 THEN S04_TargetPosition := 55; END_IF
_ft15(CLK := _S04_MovingX);
_w68 := _w67 AND (CTU_0.Q OR _ft15.Q);
S04_MX15 R= _w68;
S01_MX10 S= _w68;

END_PROGRAM
